TYPE DAQ_CTR_INTERNAL :
STRUCT
	Activate_Trigger	:DataTrigger:= 0;
	CSVWriteMode		:CSVWriteMode:=0;
	Acquire_Keyence		:BOOL		:= FALSE;
	Acquire_Massa		:BOOL		:= FALSE;
	Acquire_Sonar		:BOOL		:= FALSE;
	Keyence_Done		:BOOL		:= FALSE;
	Massa_Done			:BOOL		:= FALSE;
	Sonar_Done			:BOOL		:= FALSE;
	Clear_X				:BOOL;
	Clear_Y				:BOOL;
	Clear_Z				:BOOL;
	Clear_Time			:BOOL;
	Clear_Massa			:BOOL;
	Clear_Keyence		:BOOL;
	Clear_DAQ_Task		:BOOL;
	
	Measure_Run_Time	:BOOL		:= FALSE;
	
	Write_Data			:BOOL;
	Write_Data_Append	:BOOL;
END_STRUCT
END_TYPE

(* stored: Version 1.1.0.1, ProductVersion 3.1.4026.12
   DUT DAQ_CTR_INTERNAL: Id {93e6dfdc-3ddc-473a-813a-4c15b2117c92} *)
